(* IEC 61131-3 sources: Substation-Feeder-Automation/plc, 2 files *)

(* ---- Heartbeat.st ---- *)
PROGRAM Heartbeat
VAR
    {attribute 'symbol' := 'read'}
    Counter : UDINT := 0;
    PulseTimer : TON;
    CommandTimer : TON;
END_VAR

// Called after PLC_PRG in the same MainTask.
// Increment every ~500 ms. Explicit wrap avoids overflow exceptions.
PulseTimer(IN := NOT PulseTimer.Q, PT := T#500ms);
IF PulseTimer.Q THEN
    IF Counter >= UDINT#4294967295 THEN
        Counter := 0;
    ELSE
        Counter := Counter + 1;
    END_IF;
END_IF;

// Lab HMI command duration guard. This POU runs after PLC_PRG.
// Independent of browser/Gateway cleanup; outputs recompute next 20 ms scan.
CommandTimer(IN := PLC_PRG.Cmd_CB_Open OR PLC_PRG.Cmd_CB_Close, PT := T#7s);
IF CommandTimer.Q THEN
    PLC_PRG.Cmd_CB_Open := FALSE;
    PLC_PRG.Cmd_CB_Close := FALSE;
END_IF;

(* ---- PLC_PRG.declaration.st ---- *)
PROGRAM PLC_PRG
VAR

    {attribute 'symbol' := 'readwrite'}
    Mode_Remote             : BOOL := TRUE;
    {attribute 'symbol' := 'readwrite'}
    Sts_DC_Healthy          : BOOL := TRUE;
    {attribute 'symbol' := 'readwrite'}
    Sts_Protection_Healthy  : BOOL := TRUE;
    {attribute 'symbol' := 'readwrite'}
    Sts_CB_Open             : BOOL := TRUE;
    {attribute 'symbol' := 'readwrite'}
    Sts_BusDS_Closed        : BOOL := TRUE;
    {attribute 'symbol' := 'readwrite'}
    Sts_LineDS_Closed       : BOOL := TRUE;
    {attribute 'symbol' := 'readwrite'}
    Sts_GroundDS_Open       : BOOL := TRUE;
    {attribute 'symbol' := 'readwrite'}
    Sts_Lockout86           : BOOL := FALSE;

    {attribute 'symbol' := 'read'}
    Perm_CB_Close           : BOOL := FALSE;
    {attribute 'symbol' := 'read'}
    Out_CB_Close            : BOOL := FALSE;
    {attribute 'symbol' := 'read'}
    Out_CB_Open             : BOOL := FALSE;
END_VAR
VAR_INPUT
    {attribute 'symbol' := 'readwrite'}
	Cmd_CB_Close            : BOOL := FALSE;
    {attribute 'symbol' := 'readwrite'}
    Cmd_CB_Open             : BOOL := FALSE;
END_VAR
